FUNCTION_BLOCK TListOfEventHandlers
VAR
    Handlers : ARRAY[0..Parameters.MaxHandlers] OF IEventHandlerBase;
    HandlerCount : DINT;
END_VAR

METHOD AddHandler : BOOL
VAR_INPUT
    Handler : IEventHandlerBase;
END_VAR
IF HandlerCount < Parameters.MaxHandlers THEN
    Handlers[HandlerCount] := Handler;
    HandlerCount := HandlerCount + 1;
    AddHandler := TRUE;
END_IF
END_METHOD

METHOD Clear
VAR_INPUT
END_VAR
F_ClearMem(Handlers);
HandlerCount := 0;
END_METHOD

PROPERTY Count : DINT
GET
Count := HandlerCount;
END_GET
END_PROPERTY

METHOD GetHandler : IEventHandlerBase
VAR_INPUT
    Index : DINT;
END_VAR
IF Index < HandlerCount AND Index >= 0 THEN 
    GetHandler := Handlers[Index];
END_IF
END_METHOD

END_FUNCTION_BLOCK

(* stored: Version 1.1.0.1, ProductVersion 3.1.4024.3
   POU TListOfEventHandlers: Id {85f14c8b-0ca5-47ce-99e5-15e5f446cd3d}, SpecialFunc None
   Method AddHandler: Id {e235082a-c1d7-4854-999a-941a93196dcb}
   Method Clear: Id {517bde54-a08c-4765-8360-83de883795bf}
   Property Count: Id {051c0e08-e2d2-40b5-b383-8c8967d01b1e}
   Get Get: Id {27aa9bef-5572-4975-8c54-e9936c87f5b5}
   Method GetHandler: Id {7ee089ca-859e-40ec-b47d-6295f5fb4514} *)
